{attribute 'qualified_only'}
{attribute 'strict'}
{attribute 'to_string'}
TYPE cPuckSide :
(
	None := 0,
	Clean,
	Dirty
);
END_TYPE

(* stored: Version 1.1.0.1, ProductVersion 3.1.4024.6
   DUT cPuckSide: Id {b480ef45-0ea1-4461-b556-f13f873b6e3d} *)
